GLOBALCONSTANTS AID_BO (* Button object attribute ids *)
  (* Standard: 61499-1; Description: Copyright (c) 2023 HR Agrartechnik GmbH This program and the accompanying materials are made available under the terms of the Eclipse Public License 2.0 which is available at https://www.eclipse.org/legal/epl-2.0/ SPDX-License-Identifier: EPL-2.0 *)
  (* Version 1.0, 2026-06-20, Franz Höpfinger, HR Agrartechnik GmbH *)
  PACKAGE isobus::UT::Q::const::AID;
  VAR_GLOBAL CONSTANT
    WIDTH : USINT := USINT#1; (* 1: AID_BO_WIDTH - Width in pixels. *)
    HEIGHT : USINT := USINT#2; (* 2: AID_BO_HEIGHT - Height in pixels. *)
    BACKGROUND_COLOUR : USINT := USINT#3; (* 3: AID_BO_BACKGROUND_COLOUR - Background colour index. *)
    BORDER_COLOUR : USINT := USINT#4; (* 4: AID_BO_BORDER_COLOUR - Border colour index. *)
    KEY_CODE : USINT := USINT#5; (* 5: AID_BO_KEY_CODE - Key code. *)
    OPTIONS : USINT := USINT#6; (* 6: AID_BO_OPTIONS - Bitmask: Bit 0=latchable, Bit 1=state (0=released, 1=latched), Bit 2=suppress *)
  END_VAR
END_GLOBALCONSTANTS
